PROGRAM alarm_manager
VAR
	critical_alarm_active: BOOL;
	error_alarm_active: BOOL;
	warning_alarm_active: BOOL;
END_VAR

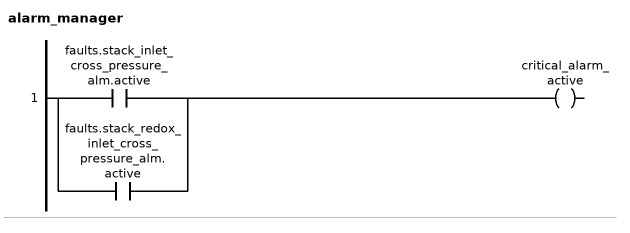
// NETWORK 1
critical_alarm_active := faults.stack_inlet_cross_pressure_alm.active OR faults.stack_redox_inlet_cross_pressure_alm.active;

END_PROGRAM

(* stored: Version 1.1.0.1, ProductVersion 3.1.4024.12
   POU alarm_manager: Id {28e37b28-da5c-4579-a648-0b987d9907b7}, SpecialFunc None *)
